% RSLogix 500 project mode,funtions.RSS, saved by version 8.30.00.16 %
PROJECT "UNTITLED"    % processor: Bul.1763 MicroLogix 1100 Series B %

PROGRAM FILES
  LAD 2 "MAIN"  2 rungs
  LAD 3 "I/O"  10 rungs

DATA FILES
  O0 OUTPUT  4 elements
  I1 INPUT  6 elements
  S2 STATUS  66 elements
  B3 BINARY  1 elements
  T4 TIMER  4 elements
  C5 COUNTER  5 elements
  R6 CONTROL  1 elements
  N7 INTEGER  4 elements
  F8 FLOAT  1 elements
  ST9   7 elements

LADDER 2 "MAIN"
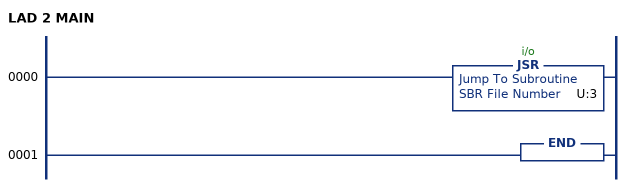
% Rung: 0 %
SOR JSR U:3 EOR
%   U:3  "i/o" %
% Rung: 1 %
SOR END EOR

LADDER 3 "I/O"
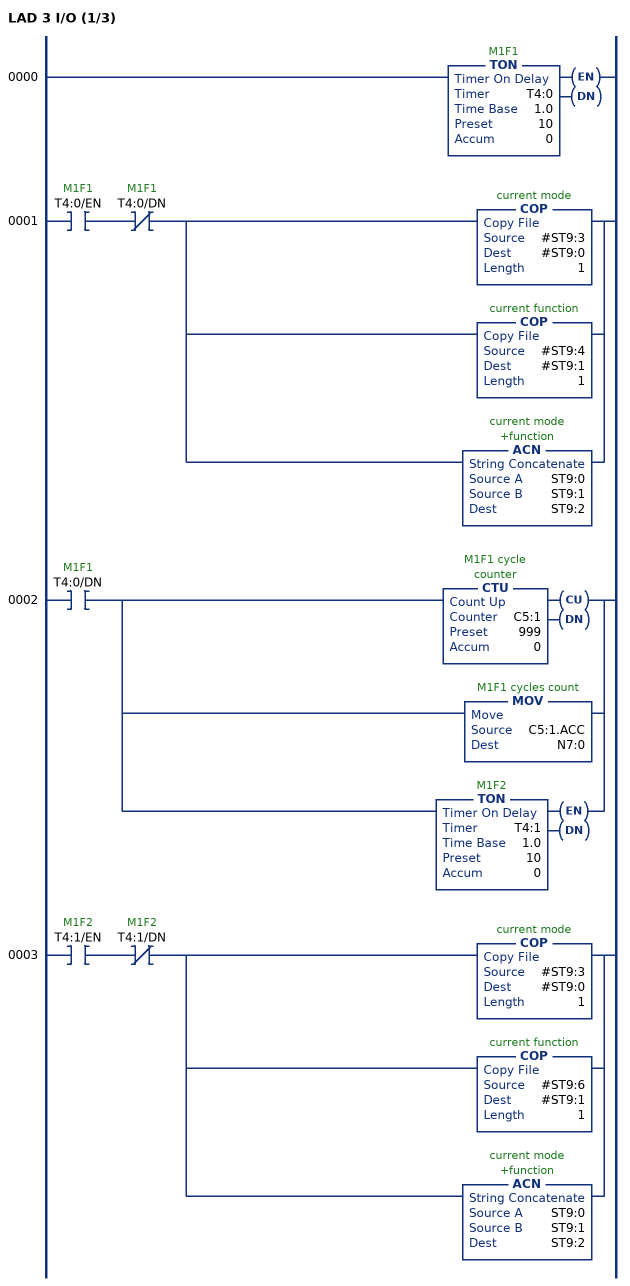
% Rung: 0 %
SOR TON T4:0 1.0 10 0 EOR
%   T4:0  "M1F1" %
% Rung: 1 %
SOR XIC T4:0/EN XIO T4:0/DN BST COP #ST9:3 #ST9:0 1 NXB COP #ST9:4 #ST9:1 1 NXB ACN ST9:0 ST9:1 ST9:2 BND EOR
%   T4:0  "M1F1" %
%   ST9:3  "MODE 1" %
%   ST9:0  "current mode" %
%   ST9:4  "FUN 1" %
%   ST9:1  "current function" %
%   ST9:2  "current mode +function" %
% Rung: 2 %
SOR XIC T4:0/DN BST CTU C5:1 999 0 NXB MOV C5:1.ACC N7:0 NXB TON T4:1 1.0 10 0 BND EOR
%   T4:0  "M1F1" %
%   C5:1  "M1F1 cycle counter" %
%   N7:0  "M1F1 cycles count" %
%   T4:1  "M1F2" %
% Rung: 3 %
SOR XIC T4:1/EN XIO T4:1/DN BST COP #ST9:3 #ST9:0 1 NXB COP #ST9:6 #ST9:1 1 NXB ACN ST9:0 ST9:1 ST9:2 BND EOR
%   T4:1  "M1F2" %
%   ST9:3  "MODE 1" %
%   ST9:0  "current mode" %
%   ST9:6  "FUN 2" %
%   ST9:1  "current function" %
%   ST9:2  "current mode +function" %

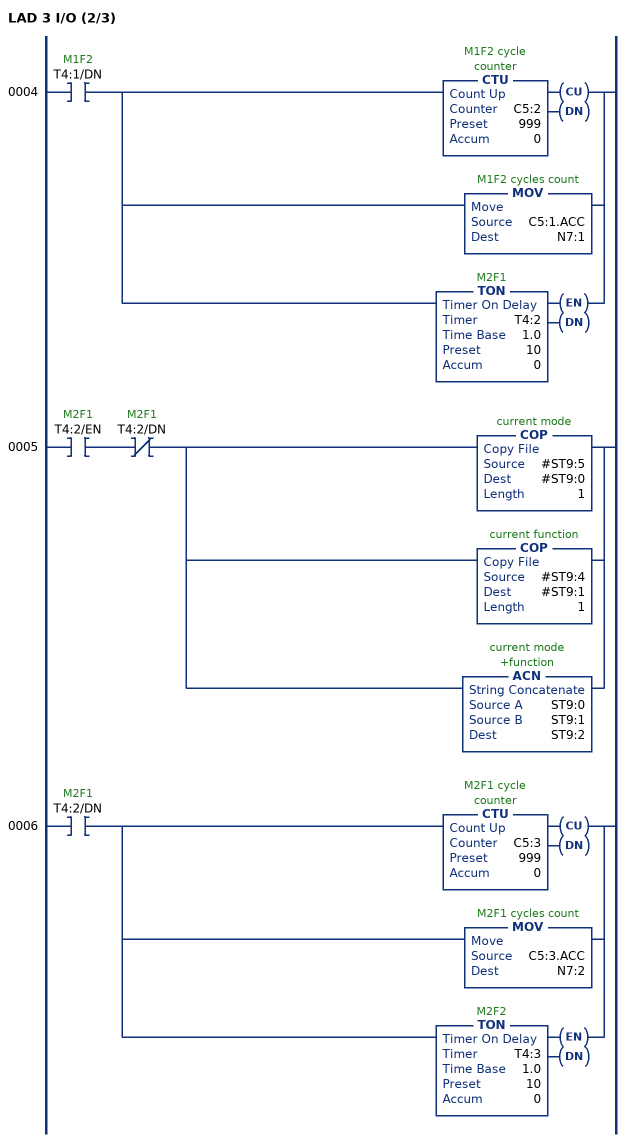
% Rung: 4 %
SOR XIC T4:1/DN BST CTU C5:2 999 0 NXB MOV C5:1.ACC N7:1 NXB TON T4:2 1.0 10 0 BND EOR
%   T4:1  "M1F2" %
%   C5:2  "M1F2 cycle counter" %
%   C5:1  "M1F1 cycle counter" %
%   N7:1  "M1F2 cycles count" %
%   T4:2  "M2F1" %
% Rung: 5 %
SOR XIC T4:2/EN XIO T4:2/DN BST COP #ST9:5 #ST9:0 1 NXB COP #ST9:4 #ST9:1 1 NXB ACN ST9:0 ST9:1 ST9:2 BND EOR
%   T4:2  "M2F1" %
%   ST9:5  "MODE 2" %
%   ST9:0  "current mode" %
%   ST9:4  "FUN 1" %
%   ST9:1  "current function" %
%   ST9:2  "current mode +function" %
% Rung: 6 %
SOR XIC T4:2/DN BST CTU C5:3 999 0 NXB MOV C5:3.ACC N7:2 NXB TON T4:3 1.0 10 0 BND EOR
%   T4:2  "M2F1" %
%   C5:3  "M2F1 cycle counter" %
%   N7:2  "M2F1 cycles count" %
%   T4:3  "M2F2" %

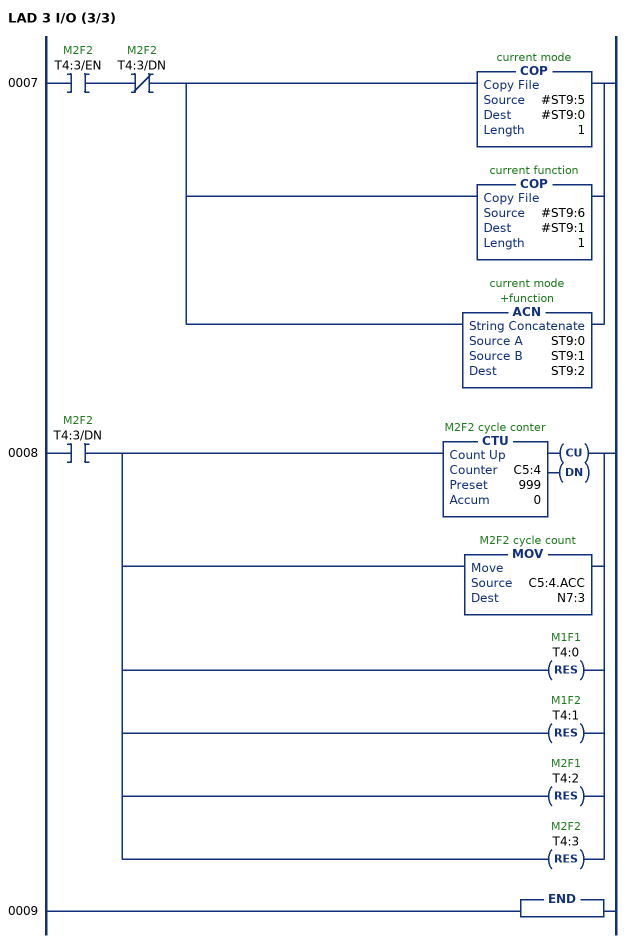
% Rung: 7 %
SOR XIC T4:3/EN XIO T4:3/DN BST COP #ST9:5 #ST9:0 1 NXB COP #ST9:6 #ST9:1 1 NXB ACN ST9:0 ST9:1 ST9:2 BND EOR
%   T4:3  "M2F2" %
%   ST9:5  "MODE 2" %
%   ST9:0  "current mode" %
%   ST9:6  "FUN 2" %
%   ST9:1  "current function" %
%   ST9:2  "current mode +function" %
% Rung: 8 %
SOR XIC T4:3/DN BST CTU C5:4 999 0 NXB MOV C5:4.ACC N7:3 NXB RES T4:0 NXB RES T4:1 NXB RES T4:2 NXB RES T4:3 BND EOR
%   T4:3  "M2F2" %
%   C5:4  "M2F2 cycle conter" %
%   N7:3  "M2F2 cycle count" %
%   T4:0  "M1F1" %
%   T4:1  "M1F2" %
%   T4:2  "M2F1" %
% Rung: 9 %
SOR END EOR

OTHER DOCUMENTED ADDRESSES
  B3:0/0  RESET_BUTTON
  B3:0/1  "reset trigger"

DATA TABLE (non-zero values as saved)
DATA T4
% .PRE .ACC %
% T4:0 % 10 0
% T4:1 % 10 0
% T4:2 % 10 0
% T4:3 % 10 0
DATA C5
% .PRE .ACC %
% C5:1 % 999 0
% C5:2 % 999 0
% C5:3 % 999 0
% C5:4 % 999 0
DATA ST9
% ST9:3 % "MODE1"
% ST9:4 % "FUN1"
% ST9:5 % "MODE2"
% ST9:6 % "FUN2"
